{attribute 'GeneratedUsingTerminal: EPP1816-0008-0016'}
{attribute addProperty BoxType "EPP1816-0008-0016"}
{attribute addProperty Id "EtcSlaveTerminalBaseDIG_Inputs_Channel_1AT %I*DIG_Inputs_Channel_CC4551489DIG_Inputs_Channel_2AT %I*DIG_Inputs_Channel_CC4551489WcStateAT %I*WcState_9091E0EB2InfoDataAT %I*InfoData_32EB74EA10"}
{attribute addProperty CRC "1648857749"}
{attribute addProperty Size "30"}
TYPE EPP1816_62479295 EXTENDS EtcSlaveTerminalBase :
STRUCT
	{attribute addProperty Name "DIG_Inputs_Channel_1"}
	DIG_Inputs_Channel_1 : DIG_Inputs_Channel_CC455148;
	{attribute addProperty Name "DIG_Inputs_Channel_2"}
	DIG_Inputs_Channel_2 : DIG_Inputs_Channel_CC455148;
	{attribute addProperty Name "WcState"}
	WcState : WcState_9091E0EB;
	{attribute addProperty Name "InfoData"}
	InfoData : InfoData_32EB74EA;
END_STRUCT
END_TYPE

(* stored: Version 1.2.0.0, ProductVersion 3.1.4024.9
   DUT EPP1816_62479295: Id {c41f104c-d787-43ba-8174-56ff6d12c54f} *)
